# EPICS substitutions: iocBoot/iocvxWorks/asynRecord.substitutions
file "$(ASYN)/db/asynRecord.db"
{
pattern
{P        R         PORT    ADDR    OMAX  IMAX}
{CARS:     asyn_1   serial1    0     256  256}
{CARS:     asyn_2   serial2    0     256  256}
{CARS:     asyn_3   serial3    0     256  256}
{CARS:     asyn_4   serial4    0     256  256}
{CARS:     asyn_5   serial5    0     256  256}
{CARS:     asyn_6   serial6    0    2600  2600}
{CARS:     asyn_7   serial7    0     256  256}
{CARS:     asyn_8   serial8    0     256  256}
#{CARS:     gpib1    gpib1      1    2600 2600}
}
